FUNCTION_BLOCK StateList
VAR_GENERIC CONSTANT
	MaxCount : DINT := 10;
END_VAR IMPLEMENTS I_StateList
VAR
	States : ARRAY[0..MaxCount] OF I_State;
END_VAR

METHOD AddStateAtIndex
VAR_INPUT
	Index : DINT;
	State : I_State;
END_VAR
IF Index > MaxCount THEN
	RETURN;
END_IF

States[Index] := State;
END_METHOD

METHOD GetStateAtIndex : I_State
VAR_INPUT
	Index : DINT;
END_VAR
IF Index > MaxCount THEN
	RETURN;
END_IF

GetStateAtIndex := States[Index];
END_METHOD

PROPERTY NumberOfStates : DINT
GET
NumberOfStates := MaxCount;
END_GET
END_PROPERTY

END_FUNCTION_BLOCK

(* stored: Version 1.1.0.1, ProductVersion 3.1.4026.18
   POU StateList: Id {b9677d1f-46db-46ec-81b0-8c3821098953}, SpecialFunc None
   Method AddStateAtIndex: Id {5c241dee-4946-49cf-95b8-783756096cf4}
   Method GetStateAtIndex: Id {45de4b0b-2e2d-4f8a-9529-30ab85ff8fac}
   Property NumberOfStates: Id {d6a3c2b0-4380-46a5-beaf-abe63d9022e0}
   Get Get: Id {970c706a-78c3-4730-8137-2fbd69e4719d} *)
